INTERFACE ITF_MessengerRecipient

END_INTERFACE

(* stored: Version 1.1.0.1
   Itf ITF_MessengerRecipient: Id {79cc86b5-6733-0d7e-064a-2560a6148741} *)
